TYPE ST_Arg :
STRUCT
	eType : E_ArgType			:= E_ArgType.VoidArg;
	pData : POINTER TO BYTE		:= 0;
	nSize : BYTE				:= 0;
END_STRUCT
END_TYPE

(* stored: Version 1.1.0.1, ProductVersion 3.1.4024.15
   DUT ST_Arg: Id {f634bd9d-7348-4622-9698-a3bf22d45288} *)
